//=============================================================================
// FB_StateMachine
//-----------------------------------------------------------------------------
// Core sequencer, ported from the DirectSoft6 ISG/SG stage flow (S0..S13).
// One CASE statement = one place state can ever change.
//
// External events arrive through the Request*() methods (called by MAIN from
// FB_Hmi command pulses). The methods only SET request flags; the actual
// transition happens inside the CASE so ordering is deterministic and a
// request can be validated/refused in one spot.
//
// Outputs are "enable" flags consumed by the control FBs and FB_OutputHandler.
// This FB never writes I/O directly.
//
// Transition map (verified against the JMP instructions in the source):
//   ControllerInit -> SesOff
//   SesOff -> CheckIfHot            (start requested, no blocking fault)
//   CheckIfHot -> SteamFlowing      (C14: SPA warm AND flow > 5%  -> hot restart)
//              -> InitFillWater      (cold, drain bit C30 clear)
//   InitFillWater -> InitPurgeVessel (fill complete)
//                 -> SesOff          (abort)
//   InitPurgeVessel -> InitSetDiffPressure (purge complete)
//                   -> SesOff / Fault
//   InitSetDiffPressure -> InitMain  (dP established within T13)
//                       -> Fault      (downstream start-high / timeout)
//   InitMain -> SteamFlowing          (init complete)
//            -> SesOff                 (abort)
//   SteamFlowing -> SesOff             (stop requested)
//   Maintenance  -> SesOff             (exit)
//   Fault -> ControllerInit            (operator reset ONLY)
//   (any startup/run state) -> Maintenance  (maint requested from SesOff only)
//=============================================================================
FUNCTION_BLOCK FB_StateMachine_1
VAR_INPUT
    stProcess   : ST_ProcessValues;
    stFaults    : ST_Faults;
    stSetpoints : ST_HmiSetpoints;
END_VAR
VAR_OUTPUT
    eState           : E_SystemState := E_SystemState.ControllerInit;

    // enable flags for downstream FBs
    bControlEnable   : BOOL;   // PID pressure/temp loops may run
    bWaterFillEnable : BOOL;   // water fill sequence active
    bPurgeEnable     : BOOL;   // vessel purge sequence active
    bReady           : BOOL;   // green Ready: in SteamFlowing, in-band, no faults

    bInStartup       : BOOL;   // TRUE for any Init* state (HMI "starting..." hint)
END_VAR
VAR
    // --- request flags set by methods, cleared when serviced ---
    bReqStart        : BOOL;
    bReqStop         : BOOL;
    bReqMaint        : BOOL;
    bReqExitMaint    : BOOL;
    bReqFault        : BOOL;
    bReqFaultReset   : BOOL;

    // --- state entry detection (rising edge of a new state) ---
    eStatePrev       : E_SystemState;
    bEntry           : BOOL;   // TRUE on the first cycle of the current state

    // --- per-state timers (replaces legacy T11 warmup, T13 dP, etc.) ---
    tonWarmup        : TON;    // TC3 warmup, legacy 120 s (V1532)
    tonDiffPress     : TON;    // dP settle, legacy 15 min baseline (see rung ~498)
    tonFillTimeout   : TON;
    tonPurgeTimeout  : TON;

    // --- thresholds (seed from GVL_Params at init; defaults from source) ---
    tWarmupTime      : TIME := T#120S;   // legacy "Begin a 120 sec warm up timer for TC3"
    tDiffPressTime   : TIME := T#15M;    // legacy baseline 15 min
    tFillTimeout     : TIME := T#10M;
    tPurgeTimeout    : TIME := T#10M;
    rHotRestartFlowPct : REAL := 5.0;    // legacy "steam flow is over 5%"
END_VAR

//=========================== entry-edge detection =============================
bEntry := (eState <> eStatePrev);
eStatePrev := eState;

//=========================== global fault override ===========================
// A latching fault forces Fault from ANY state except when already resetting.
// This mirrors the ~25 scattered "JMP S10" checks in the source, now funneled
// through one request from FB_FaultMonitor (see MAIN).
IF bReqFault AND (eState <> E_SystemState.Fault) THEN
    eState := E_SystemState.Fault;
    bEntry := TRUE;
END_IF
bReqFault := FALSE;

//=========================== default enable flags ============================
// Recomputed every cycle; each state turns on what it needs below.
bControlEnable   := FALSE;
bWaterFillEnable := FALSE;
bPurgeEnable     := FALSE;
bReady           := FALSE;
bInStartup       := FALSE;

//================================ STATE MACHINE ==============================
CASE eState OF

    //--------------------------------------------------------------------
    E_SystemState.ControllerInit:   // S0 : one-shot init, then idle
    //--------------------------------------------------------------------
        // Most legacy S0 param-loads are now variable initializers / PERSISTENT.
        // Nothing to hold here; drop straight to idle once entry housekeeping
        // is done.
        IF bEntry THEN
            // TODO: seed thresholds from GVL_Params here if they differ per unit
            ;
        END_IF
        eState := E_SystemState.SesOff;

    //--------------------------------------------------------------------
    E_SystemState.SesOff:           // S6 : idle / standby
    //--------------------------------------------------------------------
        // Legacy: "Reset warmup timer while in SES OFF" (rung ~1978)
        tonWarmup(IN := FALSE);

        IF bReqMaint THEN
            eState := E_SystemState.Maintenance;
        ELSIF bReqStart AND NOT stFaults.bHmiCommLoss THEN
            eState := E_SystemState.CheckIfHot;
        END_IF

    //--------------------------------------------------------------------
    E_SystemState.CheckIfHot:       // S101 : hot-restart shortcut vs cold start
    //--------------------------------------------------------------------
        // Legacy C14 (rung 84): SPA warm (TC1 within band V1505..V1507)
        // AND steam flow already > 5% -> jump straight to SteamFlowing.
        // Otherwise cold start -> fill water (drain bit C30 clear).
        bInStartup := TRUE;
        IF _IsSpaWarm() AND (_FlowPercent() > rHotRestartFlowPct) THEN
            eState := E_SystemState.SteamFlowing;   // legacy: SET Y2, JMP S4
        ELSE
            eState := E_SystemState.InitFillWater;  // legacy: JMP S111
        END_IF

    //--------------------------------------------------------------------
    E_SystemState.InitFillWater:    // S111 : fill water
    //--------------------------------------------------------------------
        bInStartup       := TRUE;
        bWaterFillEnable := TRUE;
        tonFillTimeout(IN := TRUE, PT := tFillTimeout);

        IF bReqStop THEN
            eState := E_SystemState.SesOff;
        ELSIF stFaults.bWaterFill OR tonFillTimeout.Q THEN
            bReqFault := TRUE;   // serviced top-of-cycle next scan
        ELSIF stProcess.bWaterFull THEN            // fill complete
            eState := E_SystemState.InitPurgeVessel;
        END_IF

    //--------------------------------------------------------------------
    E_SystemState.InitPurgeVessel:  // S11 : purge vessel
    //--------------------------------------------------------------------
        bInStartup   := TRUE;
        bPurgeEnable := TRUE;
        tonPurgeTimeout(IN := TRUE, PT := tPurgeTimeout);

        IF bReqStop THEN
            eState := E_SystemState.SesOff;
        ELSIF stFaults.bVesselPurge OR tonPurgeTimeout.Q THEN
            bReqFault := TRUE;
        ELSIF stProcess.bSpaFlushed THEN           // purge complete
            eState := E_SystemState.InitSetDiffPressure;
        END_IF

    //--------------------------------------------------------------------
    E_SystemState.InitSetDiffPressure: // S13 : establish differential pressure
    //--------------------------------------------------------------------
        bInStartup     := TRUE;
        bControlEnable := TRUE;   // dP PID runs to bring differential up
        tonDiffPress(IN := TRUE, PT := tDiffPressTime);

        IF stFaults.bDownstreamStartHigh OR stFaults.bStartupDiffPress THEN
            bReqFault := TRUE;    // legacy DS start-high -> S10
        ELSIF tonDiffPress.Q THEN
            bReqFault := TRUE;    // could not establish dP in time
        ELSIF _IsDiffPressEstablished() THEN
            eState := E_SystemState.InitMain;
        END_IF

    //--------------------------------------------------------------------
    E_SystemState.InitMain:         // S1 : final checks before flow
    //--------------------------------------------------------------------
        bInStartup     := TRUE;
        bControlEnable := TRUE;

        IF bReqStop THEN
            eState := E_SystemState.SesOff;
        ELSIF _IsInitComplete() THEN
            eState := E_SystemState.SteamFlowing;
        END_IF

    //--------------------------------------------------------------------
    E_SystemState.SteamFlowing:     // S4 : normal production
    //--------------------------------------------------------------------
        bControlEnable := TRUE;
        // Ready = producing, no active faults, flow tracking setpoint
        bReady := NOT stFaults.bHmiCommLoss
                  AND _FlowInBand()
                  AND _TempsInBand();

        IF bReqStop THEN
            eState := E_SystemState.SesOff;
        END_IF

    //--------------------------------------------------------------------
    E_SystemState.Maintenance:      // S7 : manual actuation
    //--------------------------------------------------------------------
        // Outputs handled by FB_OutputHandler via HMI overrides; no auto control.
        IF bReqExitMaint OR bReqStop THEN
            eState := E_SystemState.SesOff;
        END_IF

    //--------------------------------------------------------------------
    E_SystemState.Fault:            // S10 : latched fault
    //--------------------------------------------------------------------
        // All auto outputs off. Only an operator reset leaves this state,
        // and only once all latching faults have actually cleared.
        IF bReqFaultReset AND NOT stFaults.bHmiCommLoss THEN
            eState := E_SystemState.ControllerInit;   // legacy S10 -> S0
        END_IF

ELSE
    // Unknown/illegal state -> safe fallback
    eState := E_SystemState.Fault;
END_CASE

//=========================== clear serviced requests =========================
// (bReqFault is cleared at the top of the next cycle after being serviced.)
bReqStart      := FALSE;
bReqStop       := FALSE;
bReqMaint      := FALSE;
bReqExitMaint  := FALSE;
bReqFaultReset := FALSE;

METHOD PRIVATE _FlowInBand : BOOL
// within +/-10% of setpoint (TODO: tune / pull tolerance from params)
_FlowInBand := ABS(stProcess.rFlowActual - stSetpoints.rSetFlow)
               <= (0.10 * stSetpoints.rSetFlow);
END_METHOD

METHOD PRIVATE _FlowPercent : REAL
IF stProcess.rFlowRated > 0.0 THEN
    _FlowPercent := 100.0 * stProcess.rFlowActual / stProcess.rFlowRated;
ELSE
    _FlowPercent := 0.0;
END_IF
END_METHOD

// TODO: real dP target from setpoints/params (legacy "Purge dP"/INI_SP).
METHOD PRIVATE _IsDiffPressEstablished : BOOL
_IsDiffPressEstablished := (stProcess.rDiffPressure >= stSetpoints.rSetDsPressure);
END_METHOD

// TODO: port the final S1 readiness checks (temps settled, dP stable).
METHOD PRIVATE _IsInitComplete : BOOL
_IsInitComplete := _TempsInBand() AND _IsDiffPressEstablished();
END_METHOD

// Legacy C14 part 1: TC1 SPA within warm band (V1505..V1507).
// TODO: replace band with real values from GVL_Params.
METHOD PRIVATE _IsSpaWarm : BOOL
VAR_INPUT
END_VAR
_IsSpaWarm := (stProcess.rTc1Spa >= 30.0);  // TODO: real warm-band low limit
END_METHOD

// TODO: real temperature bands from params (Warmup Temp V1535, Max Temp V1522).
METHOD PRIVATE _TempsInBand : BOOL
_TempsInBand := (stProcess.rTc1Spa >= 30.0) AND (stProcess.rTc1Spa <= 130.0);
END_METHOD

METHOD RequestExitMaint : BOOL
bReqExitMaint := TRUE;
RequestExitMaint := TRUE;
END_METHOD

// Force Fault. Called by MAIN when FB_FaultMonitor latches a fault.
METHOD RequestFault : BOOL
bReqFault := TRUE;
RequestFault := TRUE;
END_METHOD

// Operator reset. Only leaves Fault when latching faults have cleared.
METHOD RequestFaultReset : BOOL
bReqFaultReset := TRUE;
RequestFaultReset := TRUE;
END_METHOD

// Enter Maintenance. Honored only from SesOff.
METHOD RequestMaintenance : BOOL
bReqMaint := TRUE;
RequestMaintenance := TRUE;
END_METHOD

// SES ON. Honored only from SesOff (checked in the CASE).
METHOD RequestStart : BOOL
bReqStart := TRUE;
RequestStart := TRUE;
END_METHOD

// SES OFF / abort. Honored from any running or startup state.
METHOD RequestStop : BOOL
bReqStop := TRUE;
RequestStop := TRUE;
END_METHOD

END_FUNCTION_BLOCK

(* stored: Version 1.1.0.1, ProductVersion 3.1.4026.18
   POU FB_StateMachine_1: Id {a1b2c3d4-0012-4a5b-9c8d-e1f200000012}, SpecialFunc None
   Method _FlowInBand: Id {a1b2c3d4-0012-4a5b-9c8d-e1f200000205}
   Method _FlowPercent: Id {a1b2c3d4-0012-4a5b-9c8d-e1f200000202}
   Method _IsDiffPressEstablished: Id {a1b2c3d4-0012-4a5b-9c8d-e1f200000203}
   Method _IsInitComplete: Id {a1b2c3d4-0012-4a5b-9c8d-e1f200000204}
   Method _IsSpaWarm: Id {a1b2c3d4-0012-4a5b-9c8d-e1f200000201}
   Method _TempsInBand: Id {a1b2c3d4-0012-4a5b-9c8d-e1f200000206}
   Method RequestExitMaint: Id {a1b2c3d4-0012-4a5b-9c8d-e1f200000104}
   Method RequestFault: Id {a1b2c3d4-0012-4a5b-9c8d-e1f200000105}
   Method RequestFaultReset: Id {a1b2c3d4-0012-4a5b-9c8d-e1f200000106}
   Method RequestMaintenance: Id {a1b2c3d4-0012-4a5b-9c8d-e1f200000103}
   Method RequestStart: Id {a1b2c3d4-0012-4a5b-9c8d-e1f200000101}
   Method RequestStop: Id {a1b2c3d4-0012-4a5b-9c8d-e1f200000102} *)
